TYPE ActuatorConfiguration EXTENDS BaseConfiguration:
STRUCT
	//Output
	sPusherType : STRING;
	iPusherPosition : DINT;
END_STRUCT
END_TYPE

(* stored: Version 1.1.0.1, ProductVersion 3.1.4024.9
   DUT ActuatorConfiguration: Id {da2be6a3-33e9-4253-b7f2-bd765eb11f2d} *)
